PROGRAM MAIN
VAR
	// push buttons
	StartPB: BOOL;
	StopPB: BOOL;
	ResetButton: BOOL;

	// sensors
	BottomLimitSwitch: BOOL;	
	ProxSwitch: BOOL;
	
	PistonLeftPos: BOOL;
	PistonRightPos: BOOL;
	
	// HW outputs
	
	ConveyorRun: BOOL;
	LifterUp: BOOL;
	LifterDown: BOOL;
	LifterStop: BOOL;
	
	PistonMoveLeft: BOOL;
	PistonMoveRight: BOOL;

	// Aux. objects
	rtBottomLS: R_TRIG;
	rtIndexPcb: R_TRIG;
	
	tondelayLifterUp: TON;
	tonDelay1sec: TON;
	
	rtPistonLeftReached: R_TRIG;
	ctuPistonLeftMovements: CTU;
END_VAR
VAR // added by the converter: edge detectors and wires of the graphical bodies
    _w1 : BOOL;
END_VAR

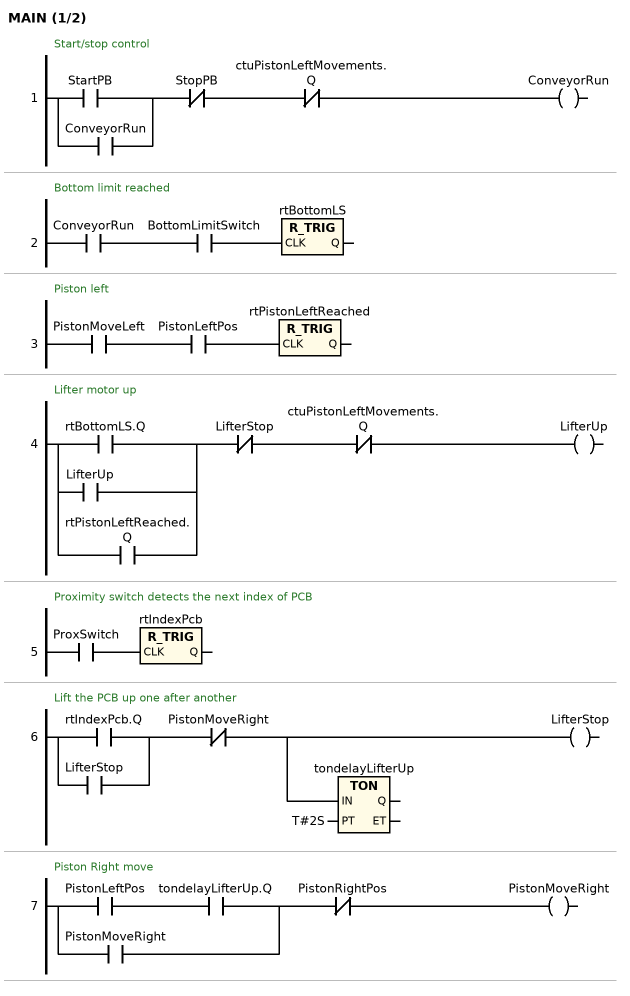
// NETWORK 1
// Start/stop control
ConveyorRun := (StartPB OR ConveyorRun) AND NOT StopPB AND NOT ctuPistonLeftMovements.Q;

// NETWORK 2
// Bottom limit reached
rtBottomLS(CLK := ConveyorRun AND BottomLimitSwitch); // R_TRIG

// NETWORK 3
// Piston left
rtPistonLeftReached(CLK := PistonMoveLeft AND PistonLeftPos); // R_TRIG

// NETWORK 4
// Lifter motor up
LifterUp := (rtBottomLS.Q OR LifterUp OR rtPistonLeftReached.Q) AND NOT LifterStop AND NOT ctuPistonLeftMovements.Q;

// NETWORK 5
// Proximity switch detects the next index of PCB
rtIndexPcb(CLK := ProxSwitch); // R_TRIG

// NETWORK 6
// Lift the PCB up one after another
_w1 := (rtIndexPcb.Q OR LifterStop) AND NOT PistonMoveRight;
LifterStop := _w1;
tondelayLifterUp(IN := _w1, PT := T#2S); // TON

// NETWORK 7
// Piston Right move
PistonMoveRight := (PistonLeftPos AND tondelayLifterUp.Q OR PistonMoveRight) AND NOT PistonRightPos;

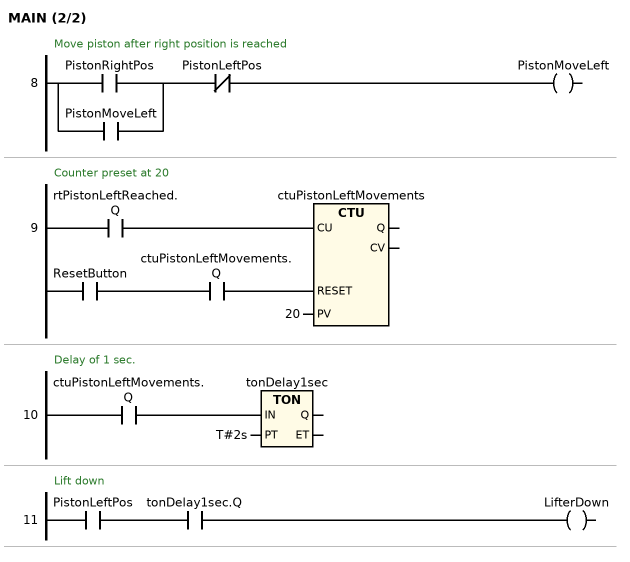
// NETWORK 8
// Move piston after right position is reached
PistonMoveLeft := (PistonRightPos OR PistonMoveLeft) AND NOT PistonLeftPos;

// NETWORK 9
// Counter preset at 20
ctuPistonLeftMovements(
    CU := rtPistonLeftReached.Q,
    RESET := ResetButton AND ctuPistonLeftMovements.Q,
    PV := 20); // CTU

// NETWORK 10
// Delay of 1 sec.
tonDelay1sec(IN := ctuPistonLeftMovements.Q, PT := T#2s); // TON

// NETWORK 11
// Lift down
LifterDown := PistonLeftPos AND tonDelay1sec.Q;

END_PROGRAM

(* stored: Version 1.1.0.1, ProductVersion 3.1.4024.15
   POU MAIN: Id {cefdf557-d300-44e0-ac30-e244246273d1}, SpecialFunc None *)
